{attribute addProperty BoxType "AT2025-0250-0022"}
{attribute addProperty Id "A_0075_AT2000_5250_0019_AT2000_5250AT2000_C5E5984862678.25"}
{attribute addProperty CRC "2635629580"}
{attribute addProperty SizeInBites "626"}
{attribute addProperty SizeInBytes "78.25"}
TYPE A_0063_AT2025_0250_0022_AT2025_0250_9D18840C EXTENDS AT2025_BA5A9548 :
STRUCT
	{attribute addProperty Name "A_0075_AT2000_5250_0019_AT2000_5250"}
	A_0075_AT2000_5250_0019_AT2000_5250 : AT2000_C5E59848;
END_STRUCT
END_TYPE

(* stored: Version 1.2.0.0, ProductVersion 3.1.4024.9
   DUT A_0063_AT2025_0250_0022_AT2025_0250_9D18840C: Id {fcd81e8b-1aef-40e3-b0f6-e86cc71b9b0e} *)
